Fanuc TP program (LS listing): _transit.ls

/PROG  _TRANSIT
/ATTR
OWNER		= MNEDITOR;
COMMENT		= "Go to Transit";
PROG_SIZE	= 277;
CREATE		= DATE 20-12-28  TIME 23:47:16;
MODIFIED	= DATE 26-06-29  TIME 14:39:10;
FILE_NAME	= ;
VERSION		= 0;
LINE_COUNT	= 6;
MEMORY_SIZE	= 757;
PROTECT		= READ_WRITE;
TCD:  STACK_SIZE	= 0,
      TASK_PRIORITY	= 50,
      TIME_SLICE	= 0,
      BUSY_LAMP_OFF	= 0,
      ABORT_REQUEST	= 0,
      PAUSE_REQUEST	= 0;
DEFAULT_GROUP	= 1,*,*,*,*;
CONTROL_CODE	= 00000000 00000000;
LOCAL_REGISTERS	= 0,0,0;
/APPL

AUTO_SINGULARITY_HEADER;
  ENABLE_SINGULARITY_AVOIDANCE   : TRUE;
/MN
   1:  !******TRASNIT TO J1 ANGLE******* ;
   2:  LBL[100] ;
   3:  PR[6,1:*Transit]=AR[1]    ;
   4:   ;
   5:J PR[6:*Transit] R[108:Transit Spd]% CNT R[109:Transit CNT]    ;
   6:  WAIT (DO[37:OFF:At Transit])    ;
/POS
/END
